FUNCTION_BLOCK S5Gate
  (* Standard: 61499-2 *)
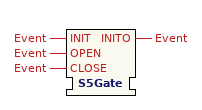
  EVENT_INPUT
    INIT;
    OPEN;
    CLOSE;
  END_EVENT
  EVENT_OUTPUT
    INITO;
  END_EVENT
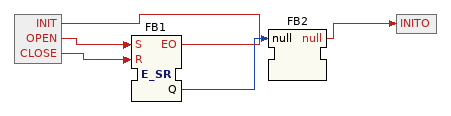
  FBS
    FB1 : E_SR;
    FB2 : ;
  END_FBS
  EVENT_CONNECTIONS
    OPEN TO FB1.S;
    CLOSE TO FB1.R;
    INIT TO FB2.null;
    FB1.EO TO FB2.null;
    FB2.null TO INITO;
  END_CONNECTIONS
  DATA_CONNECTIONS
    FB1.Q TO FB2.null;
  END_CONNECTIONS
END_FUNCTION_BLOCK
